// TIA Portal V20 export
FUNCTION_BLOCK "S7通信读写"   // FB1, LAD
{ S7_Optimized_Access := 'TRUE' }
// stored: MemoryReserve 100, SetENOAutomatically false
   VAR_INPUT
      连接ID : Word;
   END_VAR
   VAR_OUTPUT
      PUT_STATUS : Word;
      GET_STATUS : Word;
   END_VAR
   VAR_IN_OUT
      PUT_ADDR_1 : Remote;
      PUT_SD_1 : Variant;
      GET_ADDR_1 : Remote;
      GET_SD_1 : Variant;
   END_VAR
   VAR
      PUT_Instance { S7_SetPoint := 'True'} : PUT;
      GET_Instance { S7_SetPoint := 'True'} : GET;
      PUTdone : Bool;
      PUTerror : Bool;
      GETdone : Bool;
      GETerror : Bool;
   END_VAR
BEGIN

REGION Network 1
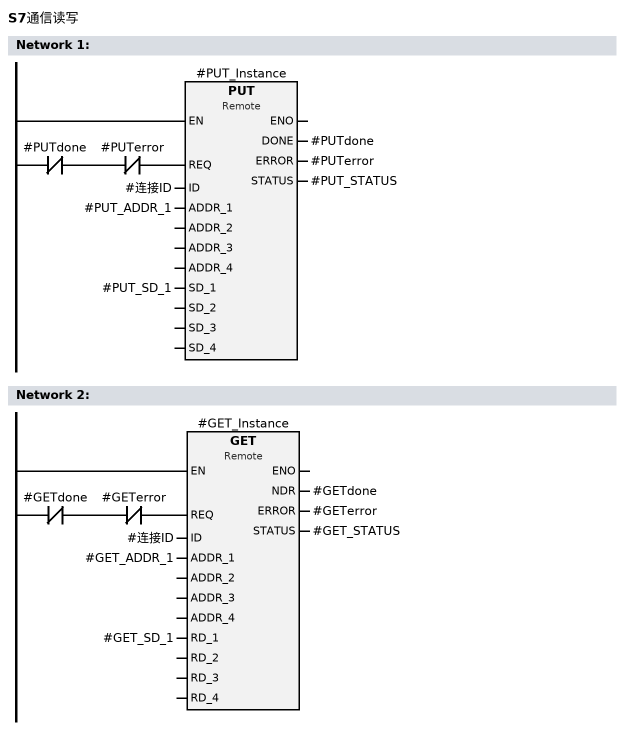
   RUNG wire#powerrail
      { S7_Templates := "[remote_type := Remote, local_type := Variant]" } #PUT_Instance.PUT(REQ := wire#w1, ID := #连接ID, ADDR_1 := #PUT_ADDR_1, ADDR_2 :=, ADDR_3 :=, ADDR_4 :=, SD_1 := #PUT_SD_1, SD_2 :=, SD_3 :=, SD_4 :=, DONE => #PUTdone, ERROR => #PUTerror, STATUS => #PUT_STATUS)
   END_RUNG
   RUNG wire#powerrail
      I_Contact( #PUTdone )
      I_Contact( #PUTerror )
   END_RUNG wire#w1
   // the same network as SCL:
   #PUT_Instance(REQ := NOT #PUTdone AND NOT #PUTerror,   // PUT
                 ID := #连接ID,
                 ADDR_1 := #PUT_ADDR_1,
                 SD_1 := #PUT_SD_1,
                 DONE => #PUTdone,
                 ERROR => #PUTerror,
                 STATUS => #PUT_STATUS);
END_REGION

REGION Network 2
   RUNG wire#powerrail
      { S7_Templates := "[remote_type := Remote, local_type := Variant]" } #GET_Instance.GET(REQ := wire#w1, ID := #连接ID, ADDR_1 := #GET_ADDR_1, ADDR_2 :=, ADDR_3 :=, ADDR_4 :=, RD_1 := #GET_SD_1, RD_2 :=, RD_3 :=, RD_4 :=, NDR => #GETdone, ERROR => #GETerror, STATUS => #GET_STATUS)
   END_RUNG
   RUNG wire#powerrail
      I_Contact( #GETdone )
      I_Contact( #GETerror )
   END_RUNG wire#w1
   // the same network as SCL:
   #GET_Instance(REQ := NOT #GETdone AND NOT #GETerror,   // GET
                 ID := #连接ID,
                 ADDR_1 := #GET_ADDR_1,
                 RD_1 := #GET_SD_1,
                 NDR => #GETdone,
                 ERROR => #GETerror,
                 STATUS => #GET_STATUS);
END_REGION
END_FUNCTION_BLOCK
